// TwinCAT 3 PLC project PLC1
// ProgramVersion: 3.1.4023.0
// libraries:
//   Tc2_Standard, * (Beckhoff Automation GmbH)
//   Tc2_System, * (Beckhoff Automation GmbH)
//   Tc3_Module, * (Beckhoff Automation GmbH)
// project tree:
//   / GlobalTextList.TcGTLO (not stored), PlcTask.TcTTO (not stored)
//   GVLs/ GVL.TcGVL
//   POUs/ MAIN.TcPOU (not stored)
// real-time tasks:
//   TASK PlcTask: cycle T#10ms, priority 20, ADS port 350

// ---- GVLs/GVL.TcGVL
{attribute 'qualified_only'}
VAR_GLOBAL
	StopButton AT %I* : BOOL;
	EmergencyStopButton AT %I* : BOOL;
	StartButton AT %I* : BOOL;
	ProductDetectedSensor AT %I* : BOOL;
	ConveyorFullSensor AT %I* : BOOL;
	MotorContactor AT %Q* : BOOL;
END_VAR
